Yaskawa INFORM job: R43_SW_OP140.JBI

/JOB
//NAME R43_SW_OP140
///FOLDERNAME JOBS
//POS
///NPOS 122,0,122,0,0,0
///TOOL 15
///POSTYPE PULSE
///PULSE
C00000=102010,-94384,-88091,-1795,-89622,-99292
C00001=108725,-63855,-97488,3358,-68955,-103488
C00002=118843,-89949,-129066,-7529,-35783,-148808
C00003=139568,-88782,-129082,65071,-35120,-199690
C00004=149969,-82921,-126695,90920,-42511,-223339
///TOOL 0
C00005=150430,-84262,-127349,90601,-43098,-223231
///TOOL 15
C00006=149969,-82921,-126695,90920,-42511,-223339
C00007=139568,-88782,-129082,65071,-35120,-199690
C00008=118843,-89949,-129066,-7529,-35783,-148808
C00009=126550,-86492,-138460,6642,-21597,-153692
C00010=130859,-86671,-139573,13597,-18453,-155898
C00011=131658,-90708,-141398,15833,-19958,-157705
///TOOL 0
C00012=131819,-91565,-141527,16072,-20472,-157919
///TOOL 15
C00013=130858,-86672,-139571,13597,-18453,-155900
C00014=117189,-85989,-147791,-63912,-14042,-97628
C00015=101892,-32658,-93105,-61319,-72428,-103505
C00016=110411,-27055,-80542,-52269,-77750,-114469
///TOOL 0
C00017=110500,-28614,-81772,-52159,-77841,-114609
///TOOL 15
C00018=110411,-27055,-80542,-52269,-77750,-114469
C00019=107141,-27026,-83463,-54792,-77046,-110769
///TOOL 0
C00020=107206,-28721,-84801,-54682,-77157,-110901
///TOOL 15
C00021=107141,-27026,-83463,-54792,-77046,-110769
C00022=101970,-27747,-88888,-58780,-75999,-104844
///TOOL 0
C00023=101966,-28750,-89865,-58815,-75954,-104813
///TOOL 15
C00024=101970,-27747,-88888,-58780,-75999,-104844
C00025=101772,-29037,-98901,-66475,-66640,-98886
C00026=108162,-25882,-97472,-68741,-63479,-101997
C00027=108246,-28047,-96196,-66583,-65474,-103876
///TOOL 0
C00028=108284,-28890,-96748,-66431,-65593,-104021
///TOOL 15
C00029=108246,-28047,-96196,-66583,-65474,-103876
C00030=109355,-32968,-111280,-85694,-51369,-87119
///TOOL 0
C00031=109535,-33757,-111980,-85596,-51282,-87277
///TOOL 15
C00032=109355,-32968,-111280,-85694,-51369,-87119
C00033=106934,-32684,-111104,-86802,-52629,-85151
C00034=110214,-31943,-108998,-69143,-50257,-95694
C00035=107293,-34185,-110074,-70062,-52189,-93685
C00036=115636,-30246,-114226,-47491,-40039,-107547
C00037=120106,-27232,-111592,-29907,-40090,-119844
C00038=129921,-23144,-107742,8794,-40346,-146950
C00039=130780,-24989,-108505,11762,-40804,-148901
///TOOL 0
C00040=130965,-26010,-109317,11966,-40908,-149135
///TOOL 15
C00041=130780,-24989,-108505,11762,-40804,-148901
C00042=119755,-28047,-112678,-43194,-38496,-112586
///TOOL 0
C00043=119927,-29549,-113839,-42826,-38593,-112934
///TOOL 15
C00044=119755,-28047,-112678,-43194,-38496,-112586
C00045=120573,-18526,-104835,-38667,-45871,-117397
C00046=123149,-17428,-104014,-36470,-45105,-120275
///TOOL 0
C00047=123228,-17946,-104561,-36439,-45032,-120331
///TOOL 15
C00048=123149,-17428,-104014,-36470,-45105,-120275
C00049=120573,-18526,-104835,-38667,-45871,-117397
C00050=111554,-20770,-106378,-45657,-48722,-107786
C00051=98446,-26103,-114391,-49959,-48722,-107786
C00052=59636,-11539,-95823,-73616,-117593,7595
C00053=59217,-27912,-69932,-67444,-142952,-6773
C00054=67640,4376,-47863,-78484,-144908,-7322
C00055=70991,5590,-46667,-79407,-143046,-8928
C00056=72873,2265,-49940,-79933,-141821,-9718
///TOOL 0
C00057=72795,861,-51525,-79944,-141696,-9564
///TOOL 15
C00058=72873,2265,-49940,-79933,-141821,-9718
C00059=74819,-24416,-65715,-83155,-130827,-13595
///TOOL 0
C00060=74771,-25795,-66969,-83152,-130857,-13575
///TOOL 15
C00061=74819,-24416,-65715,-83155,-130827,-13595
C00062=70991,5590,-46667,-79407,-143046,-8928
C00063=67640,4376,-47863,-78484,-144908,-7322
C00064=59217,-27912,-69932,-67444,-142952,-6773
C00065=125023,-76312,-89876,23064,-135075,-47188
C00066=143431,-76312,-98317,51485,-135075,-125061
C00067=181785,-54002,-138800,144490,-149141,-126842
C00068=188134,15153,-157202,144958,-156797,-138761
C00069=174683,95934,-147097,131824,-178933,-203790
C00070=180698,157462,-127618,174144,-182056,-247487
C00071=170736,165387,-114033,181513,-198859,-232971
C00072=180505,158217,-112336,175756,-190481,-231882
C00073=184281,160068,-107793,173005,-189110,-230235
///TOOL 0
C00074=184909,160261,-108475,172207,-188919,-230745
///TOOL 15
C00075=184007,159976,-107515,173349,-189191,-230019
C00076=182261,157828,-110313,174749,-189793,-230502
///TOOL 0
C00077=183231,158177,-111301,173523,-189513,-231288
///TOOL 15
C00078=182530,157924,-110591,174407,-189716,-230721
C00079=180505,158217,-112336,175756,-190481,-231882
C00080=170736,165387,-114033,181513,-198859,-232971
C00081=180698,157462,-127618,174144,-182056,-247487
C00082=185821,123184,-145317,137021,-175385,-244469
C00083=179119,98660,-132796,103099,-156895,-169934
C00084=172101,72978,-119683,67574,-137531,-91879
C00085=166734,53340,-109657,40410,-122725,-32194
C00086=163540,32019,-113864,63032,-135106,41632
C00087=147148,8818,-118159,54177,-121824,70686
C00088=113472,14300,-97277,35985,-105763,130371
C00089=90354,-9320,-92271,13190,-93176,192713
C00090=102574,30072,-49460,12752,-99653,185040
C00091=106413,47500,-23826,12171,-107523,183203
C00092=113139,49788,-21270,12096,-108499,178722
C00093=116655,39216,-34612,17240,-94707,184340
C00094=118575,33421,-41454,20501,-85911,188613
C00095=118789,30988,-44259,20629,-85493,188364
///TOOL 0
C00096=118836,30451,-44872,20656,-85406,188309
///TOOL 15
C00097=118789,30988,-44259,20629,-85493,188364
C00098=111725,32248,-46691,-5252,-79429,203296
///TOOL 0
C00099=111799,30923,-48218,-5244,-79178,203249
///TOOL 15
C00100=111725,32248,-46691,-5252,-79429,203296
C00101=118575,33421,-41454,20501,-85911,188613
C00102=116655,39216,-34612,17240,-94707,184340
C00103=113139,49788,-21270,12096,-108499,178722
C00104=118062,63104,4512,24001,-133389,173212
C00105=127978,69493,12755,42226,-144222,162507
C00106=149506,88154,15737,81253,-160661,160206
///TOOL 0
C00107=149676,87250,14429,81169,-160481,159943
///TOOL 15
C00108=149506,88154,15737,81253,-160661,160206
C00109=149301,89533,16704,81347,-160383,160186
C00110=147069,85698,14284,76877,-155591,161918
C00111=145040,83360,11130,77784,-153906,162452
C00112=145288,82426,12467,77750,-155162,163215
///TOOL 0
C00113=148570,65568,-6861,83141,-146931,152446
///TOOL 15
C00114=148425,66272,-5919,83177,-147018,152627
C00115=145288,82426,12467,77750,-155162,163215
C00116=145040,83360,11130,77784,-153906,162452
C00117=144361,80001,6457,78133,-152603,162149
C00118=143083,76944,2298,78746,-151120,162194
C00119=133461,67482,-6997,76759,-141353,166934
C00120=121434,51589,-6931,62314,-141353,166934
C00121=113416,-9637,3189,41740,-164945,182000
///TOOL 0
EC00000=53109
EC00001=53109
EC00002=54189
EC00003=54189
EC00004=54189
EC00005=793
EC00006=54189
EC00007=54189
EC00008=54189
EC00009=54189
EC00010=54189
EC00011=3737
EC00012=2120
EC00013=54189
EC00014=54189
EC00015=37372
EC00016=9343
EC00017=1255
EC00018=9343
EC00019=9343
EC00020=757
EC00021=9343
EC00022=9343
EC00023=762
EC00024=9343
EC00025=9343
EC00026=9343
EC00027=9343
EC00028=823
EC00029=9343
EC00030=9343
EC00031=519
EC00032=9343
EC00033=9343
EC00034=9343
EC00035=9343
EC00036=9343
EC00037=9343
EC00038=9343
EC00039=9343
EC00040=459
EC00041=9343
EC00042=9343
EC00043=573
EC00044=9343
EC00045=9343
EC00046=3737
EC00047=886
EC00048=3737
EC00049=37372
EC00050=37372
EC00051=37372
EC00052=37372
EC00053=37372
EC00054=29898
EC00055=29898
EC00056=9343
EC00057=358
EC00058=9343
EC00059=9343
EC00060=1283
EC00061=9343
EC00062=29898
EC00063=29898
EC00064=37372
EC00065=37372
EC00066=37372
EC00067=37372
EC00068=37372
EC00069=37372
EC00070=29898
EC00071=29898
EC00072=29898
EC00073=9343
EC00074=1487
EC00075=9343
EC00076=9343
EC00077=2006
EC00078=9343
EC00079=29898
EC00080=29898
EC00081=29898
EC00082=29898
EC00083=33670
EC00084=37620
EC00085=40640
EC00086=42205
EC00087=43466
EC00088=46057
EC00089=48723
EC00090=48723
EC00091=48723
EC00092=48723
EC00093=31514
EC00094=19613
EC00095=9343
EC00096=809
EC00097=9343
EC00098=9343
EC00099=935
EC00100=9343
EC00101=19613
EC00102=31514
EC00103=48723
EC00104=48723
EC00105=48723
EC00106=9343
EC00107=1234
EC00108=37372
EC00109=37372
EC00110=37372
EC00111=37372
EC00112=29898
EC00113=767
EC00114=9343
EC00115=29898
EC00116=37372
EC00117=37372
EC00118=37372
EC00119=37371
EC00120=37371
EC00121=37371
//INST
///DATE 2022/06/14 00:32
///ATTR SC,RW
///GROUP1 RB1,ST1
NOP
'RECUA BASCULANTE
DOUT OT#(321) OFF
DOUT OT#(322) ON
'AGUARDA POSICAO BASCULANTE
WAIT IN#(323)=ON
MOVJ C00000 EC00000 VJ=25.00
MOVJ C00001 EC00001 VJ=25.00
MOVJ C00002 EC00002 VJ=25.00
MOVJ C00003 EC00003 VJ=25.00
MOVJ C00004 EC00004 VJ=25.00 PL=2
'PT 118 (PT S/N)
SVSPOTMOV C00005 EC00005 V=600.0 CLF#(1) GUN#(1) PRESS#(23) WTM=23 WST=1
MOVJ C00006 EC00006 VJ=25.00 PL=2
MOVJ C00007 EC00007 VJ=25.00
MOVJ C00008 EC00008 VJ=25.00
MOVJ C00009 EC00009 VJ=25.00
MOVJ C00010 EC00010 VJ=25.00 PL=2
MOVJ C00011 EC00011 VJ=25.00
'PT 101 (PT 05)
SVSPOTMOV C00012 EC00012 V=600.0 CLF#(1) GUN#(1) PRESS#(21) WTM=21 WST=1
MOVJ C00013 EC00013 VJ=25.00
MOVJ C00014 EC00014 VJ=25.00
MOVJ C00015 EC00015 VJ=25.00
MOVJ C00016 EC00016 VJ=25.00
'PT 106 (PT 24)
SVSPOTMOV C00017 EC00017 V=600.0 CLF#(1) GUN#(1) PRESS#(99) WTM=99 WST=1
MOVJ C00018 EC00018 VJ=25.00
MOVJ C00019 EC00019 VJ=25.00 PL=2
'PT 107 (PT 23)
SVSPOTMOV C00020 EC00020 V=600.0 CLF#(1) GUN#(1) PRESS#(98) WTM=98 WST=1
MOVJ C00021 EC00021 VJ=25.00
MOVJ C00022 EC00022 VJ=25.00 PL=2
'PT 108 (PT 22)
SVSPOTMOV C00023 EC00023 V=600.0 CLF#(1) GUN#(1) PRESS#(96) WTM=96 WST=1
MOVJ C00024 EC00024 VJ=25.00 PL=2
MOVJ C00025 EC00025 VJ=25.00 PL=2
MOVJ C00026 EC00026 VJ=25.00
MOVJ C00027 EC00027 VJ=25.00
SVSPOTMOV C00028 EC00028 V=600.0 CLF#(1) GUN#(1) PRESS#(51) WTM=51 WST=1
'PT 105 (PT 19)
MOVJ C00029 EC00029 VJ=25.00
MOVJ C00030 EC00030 VJ=25.00 PL=2
SVSPOTMOV C00031 EC00031 V=600.0 CLF#(1) GUN#(1) PRESS#(110) WTM=110 WST=1
'PT 104 (PT 28)
MOVJ C00032 EC00032 VJ=25.00
MOVJ C00033 EC00033 VJ=25.00
MOVJ C00034 EC00034 VJ=25.00
MOVJ C00035 EC00035 VJ=25.00
MOVJ C00036 EC00036 VJ=25.00
MOVJ C00037 EC00037 VJ=25.00 PL=2
MOVJ C00038 EC00038 VJ=25.00 PL=2
MOVJ C00039 EC00039 VJ=25.00 PL=2
'PT 117 (PT S/N)
SVSPOTMOV C00040 EC00040 V=600.0 CLF#(1) GUN#(1) PRESS#(46) WTM=46 WST=1
MOVJ C00041 EC00041 VJ=25.00
EIMOVL UF#(15) C00042 EC00042 V=600.0
'PT 103 (PT 27)
SVSPOTMOV C00043 EC00043 V=600.0 CLF#(1) GUN#(1) PRESS#(45) WTM=45 WST=1
MOVJ C00044 EC00044 VJ=25.00
MOVJ C00045 EC00045 VJ=25.00
MOVJ C00046 EC00046 VJ=25.00
SVSPOTMOV C00047 EC00047 V=600.0 CLF#(1) GUN#(1) PRESS#(111) WTM=111 WST=1
'PT 102 (PT 33)
MOVJ C00048 EC00048 VJ=25.00
MOVJ C00049 EC00049 VJ=25.00
MOVJ C00050 EC00050 VJ=25.00
MOVJ C00051 EC00051 VJ=25.00
MOVJ C00052 EC00052 VJ=25.00
MOVJ C00053 EC00053 VJ=25.00
MOVJ C00054 EC00054 VJ=25.00 PL=1
MOVJ C00055 EC00055 VJ=25.00 PL=1
MOVJ C00056 EC00056 VJ=25.00
'PT 109 (PT 04)
SVSPOTMOV C00057 EC00057 V=600.0 CLF#(1) GUN#(1) PRESS#(17) WTM=17 WST=1
MOVJ C00058 EC00058 VJ=25.00
EIMOVL UF#(15) C00059 EC00059 V=600.0
'PT 110 (PT 20)
SVSPOTMOV C00060 EC00060 V=600.0 CLF#(1) GUN#(1) PRESS#(18) WTM=18 WST=1
MOVJ C00061 EC00061 VJ=25.00
MOVJ C00062 EC00062 VJ=25.00 PL=1
MOVJ C00063 EC00063 VJ=25.00 PL=1
MOVJ C00064 EC00064 VJ=25.00
MOVJ C00065 EC00065 VJ=25.00
MOVJ C00066 EC00066 VJ=25.00
MOVJ C00067 EC00067 VJ=25.00
MOVJ C00068 EC00068 VJ=25.00
MOVJ C00069 EC00069 VJ=25.00
MOVJ C00070 EC00070 VJ=25.00
MOVJ C00071 EC00071 VJ=25.00
MOVJ C00072 EC00072 VJ=25.00
EIMOVL UF#(15) C00073 EC00073 V=600.0
'PT 111 (PT 29)
SVSPOTMOV C00074 EC00074 V=600.0 CLF#(1) GUN#(1) PRESS#(90) WTM=90 WST=1
MOVJ C00075 EC00075 VJ=25.00
MOVJ C00076 EC00076 VJ=25.00
'PT 112 (PT S/N)
SVSPOTMOV C00077 EC00077 V=600.0 CLF#(1) GUN#(1) PRESS#(89) WTM=89 WST=1
MOVJ C00078 EC00078 VJ=25.00
MOVJ C00079 EC00079 VJ=25.00
MOVJ C00080 EC00080 VJ=25.00
MOVJ C00081 EC00081 VJ=25.00
MOVJ C00082 EC00082 VJ=25.00
MOVJ C00083 EC00083 VJ=25.00
MOVJ C00084 EC00084 VJ=25.00
MOVJ C00085 EC00085 VJ=25.00
MOVJ C00086 EC00086 VJ=25.00
MOVJ C00087 EC00087 VJ=25.00
MOVJ C00088 EC00088 VJ=25.00
MOVJ C00089 EC00089 VJ=25.00
MOVJ C00090 EC00090 VJ=25.00
MOVJ C00091 EC00091 VJ=25.00 PL=2
MOVJ C00092 EC00092 VJ=25.00 PL=2
MOVJ C00093 EC00093 VJ=25.00 PL=2
MOVJ C00094 EC00094 VJ=25.00 PL=2
MOVJ C00095 EC00095 VJ=25.00
'PT 113 (PT 08)
SVSPOTMOV C00096 EC00096 V=600.0 CLF#(1) GUN#(1) PRESS#(33) WTM=33 WST=1
MOVJ C00097 EC00097 VJ=25.00
EIMOVL UF#(15) C00098 EC00098 V=600.0
'PT 114 (PT 07)
SVSPOTMOV C00099 EC00099 V=600.0 CLF#(1) GUN#(1) PRESS#(32) WTM=32 WST=1
MOVJ C00100 EC00100 VJ=25.00
EIMOVL UF#(15) C00101 EC00101 V=600.0 PL=2
MOVJ C00102 EC00102 VJ=25.00 PL=2
MOVJ C00103 EC00103 VJ=25.00 PL=2
EIMOVL UF#(15) C00104 EC00104 V=600.0
EIMOVL UF#(15) C00105 EC00105 V=600.0 PL=2
EIMOVL UF#(15) C00106 EC00106 V=600.0 PL=2
'PT 115 (PT 25)
SVSPOTMOV C00107 EC00107 V=600.0 CLF#(1) GUN#(1) PRESS#(101) WTM=101 WST=1
MOVJ C00108 EC00108 VJ=25.00 PL=2
MOVJ C00109 EC00109 VJ=25.00 PL=2
MOVJ C00110 EC00110 VJ=25.00 PL=2
MOVJ C00111 EC00111 VJ=25.00 PL=2
MOVJ C00112 EC00112 VJ=25.00
'PT 116 (PT S/N)
SVSPOTMOV C00113 EC00113 V=600.0 CLF#(1) GUN#(1) PRESS#(52) WTM=52 WST=1
MOVJ C00114 EC00114 VJ=25.00 PL=2
MOVJ C00115 EC00115 VJ=25.00 PL=2
MOVJ C00116 EC00116 VJ=25.00
MOVJ C00117 EC00117 VJ=25.00 PL=2
MOVJ C00118 EC00118 VJ=25.00
MOVJ C00119 EC00119 VJ=25.00
MOVJ C00120 EC00120 VJ=25.00
MOVJ C00121 EC00121 VJ=25.00
END
